// TwinCAT 3 PLC project Main
// ProgramVersion: 3.1.4022.1
// libraries:
//   Tc2_ControllerToolbox, * (Beckhoff Automation GmbH)
//   Tc2_Standard, * (Beckhoff Automation GmbH)
//   Tc2_System, * (Beckhoff Automation GmbH)
//   Tc3_Module, * (Beckhoff Automation GmbH)
//   VisuDialogs, * (System)
// project tree:
//   DUTs/ ST_HISTORY.TcDUT, ST_POINT.TcDUT
//   / GlobalTextList.TcGTLO, PlcTask.TcTTO, Visualization Manager.TcVMO (not stored)
//   GVLs/ Global.TcGVL, Global_Constant.TcGVL
//   GVLs/IO/ IO_Inputs.TcGVL, IO_Outputs.TcGVL
//   POUs/ FB_HeaterCtrl.TcPOU, MAIN.TcPOU, UpdateHistory.TcPOU, InitPidParams.TcPOU
//   VISUs/ VIS_HEATER_CONTROL.TcVIS
// real-time tasks:
//   TASK StandardTask: cycle T#10ms, priority 1, ADS port 350
//   TASK PlcTask: cycle T#10ms, priority 20, ADS port 351
// variable links:
//   Main/Main Instance <-> Simulation/Simulation Instance
//     PlcTask Inputs/IO_Inputs.i_HtrTemp <-> PlcTask Outputs/IO_Outputs.o_HtrTemp
//     PlcTask Outputs/IO_Outputs.o_HtrON <-> PlcTask Inputs/IO_Inputs.i_HtrON
//     PlcTask Outputs/IO_Outputs.o_Restart <-> PlcTask Inputs/IO_Inputs.i_Restart

CONFIGURATION Main
    RESOURCE PLC ON TwinCAT3
        TASK PlcTask(INTERVAL := T#10ms, PRIORITY := 20);
        PROGRAM MAIN WITH PlcTask : MAIN;
    END_RESOURCE
END_CONFIGURATION

// ---- DUTs/ST_HISTORY.TcDUT
// History data
//
TYPE ST_HISTORY:
STRUCT
	
	// Members...
	arPower:       ARRAY[ 1..NUM_HISTORY_POINTS ] OF REAL; // Power history [%]
	arTemperature: ARRAY[ 1..NUM_HISTORY_POINTS ] OF REAL; // Temperature history [°C]
	arTempDiff:    ARRAY[ 1..NUM_HISTORY_POINTS ] OF REAL; // Temp. differences to setp. [°C]
	
END_STRUCT
END_TYPE

// ---- DUTs/ST_POINT.TcDUT
// Point data
//
TYPE ST_POINT:
STRUCT
	
	// Members...
	Power:       REAL; // Heating power [%]
	Temperature: REAL; // Temperature [°C]
	
END_STRUCT
END_TYPE

// ---- GVLs/Global.TcGVL
// Global members
//
VAR_GLOBAL

	// Structures...
	gstHistory: ST_HISTORY; // History data
	
	// Enums...
	gePidState: E_CTRL_STATE; // PID controller state

	// Other global members	
	gPower:    LREAL;      // Heating power [%]
	gSetpoint: REAL := 50; // Temperature setpoint [°C]
	gStepChange: REAL := 10; // Change of auto-step
	gAutoStepTimer: REAL := 0; // Auto-step timer
	gBoolAutoStep: BOOL := FALSE; //Auto-step boolean on/off for auto-step-button
	
END_VAR

// ---- GVLs/Global_Constant.TcGVL
// Global constants
//
VAR_GLOBAL CONSTANT

	// Global constants...
	NUM_HISTORY_POINTS: INT := 120; // Amount of history points
	
END_VAR

// ---- GVLs/IO/IO_Inputs.TcGVL
{attribute 'qualified_only'}
// I/O Inputs
//
VAR_GLOBAL

	// Input signals...
	i_HtrTemp AT %I*: REAL; // Heater temperature [°C]
 
END_VAR

// ---- GVLs/IO/IO_Outputs.TcGVL
{attribute 'qualified_only'}
// I/O Outputs
//
VAR_GLOBAL

	// Output signals...
	o_HtrON   AT %Q*: BOOL; // Heater to ON
	o_Restart AT %Q*: BOOL; // Restart simulation
	o_AddTemp20  AT %Q*: BOOL; // Increase temperature 20C
	o_DropTemp20 AT %Q*: BOOL; // Decrease temperature 20C
	o_AutoStep AT %Q*: BOOL; // Auto-step on/off
 
END_VAR

// ---- POUs/MAIN.TcPOU
// Application main function
//
PROGRAM MAIN
VAR

	// Function blocks...
	fbHeaterCtrl: FB_HeaterCtrl; // Heater control
	
	// Other members...
	Cntr: DINT; // Counter, visiting times
	Step: SINT; // Step counter (1...100)
	
END_VAR

// Update counter
Cntr := ( Cntr + 1 );

// Hasn't the step counter overflowed yet ?
IF Step < 100 THEN

	// Increase the step counter
	Step := ( Step + 1 );
	
// else, Maximum value reached already
ELSE

	// Restart the step counter
	Step := 1;
	
END_IF

// Call the heater control
fbHeaterCtrl( Step := Step );

// Update history
UpdateHistory( Step );

END_PROGRAM

// ---- POUs/FB_HeaterCtrl.TcPOU
// Controls the heater
//
FUNCTION_BLOCK FB_HeaterCtrl
VAR_INPUT
	
	Step: SINT; // Step counter (1...100)
	
END_VAR
VAR
	
	// Function blocks...
	fbPID: FB_CTRL_PID; // PID controller
	
	// Structures...
	stParams: ST_CTRL_PID_PARAMS; // PID controller parameters
	
	// Booleans...
	bInitialized: BOOL; // Initialized
	bRestart:     BOOL; // Restart
	bAutoStep:    BOOL; // Auto-step
	
END_VAR

// Initialize members
bRestart    := ( bRestart    OR IO_Outputs.o_Restart );

// First visit ? 
IF NOT bInitialized THEN
	
	// Initialize PID controller parameters
	bInitialized := TRUE;
	InitPidParams( ADR( stParams ));
	
	bAutoStep := FALSE;
	
END_IF

// Is the the starting step ?
IF Step = 1 THEN
  
	// Update the PID controller once per every second
	fbPID
	(
		fSetpointValue := gSetpoint,
		fActualValue   := IO_Inputs.i_HtrTemp,
		fManSyncValue  := 0,
		bSync          := FALSE,
		eMode          := SEL( bRestart, eCTRL_MODE_ACTIVE, eCTRL_MODE_RESET ),
		bHold          := FALSE,
		stParams       := stParams,
		fOut           => gPower,
		eState         => gePidState
(*
		bARWactive     => BOOL;
		eErrorId       => E_CTRL_ERRORCODES;
		bError         => BOOL;
*)
	);

	// Control the heater to ON/OFF
	IO_Outputs.o_HtrON := ( fbPID.fOut >= Step );
	bRestart           := FALSE;
	
	// Auto-step control
	IF bAutoStep THEN
		gAutoStepTimer := gAutoStepTimer+1;
		IF (gAutoStepTimer >= 20) THEN
			gSetpoint := gSetpoint + gStepChange;
			IF (gSetpoint > 200) THEN
				gSetpoint := 190;
				gStepChange := -10;
			ELSIF (gSetpoint < 0) THEN
				gSetpoint := 10;
				gStepChange := 10;
			END_IF
			gAutoStepTimer := 0;
		END_IF
	END_IF
	
// else, Not the first step now => Is heater controlled to ON ?
ELSIF IO_Outputs.o_HtrON THEN
	
	// Control the heater to ON/OFF
	IO_Outputs.o_HtrON := ( fbPID.fOut >= Step );
	
END_IF

IF IO_Outputs.o_AddTemp20 THEN
	
	gSetpoint := gSetpoint + 20;
	
	IF (gSetpoint > 200) THEN
		gSetpoint := 200;
	END_IF
	
	IO_Outputs.o_AddTemp20 :=FALSE;
	
END_IF

IF IO_Outputs.o_DropTemp20 THEN
	
	gSetpoint := gSetpoint - 20;
	
	IF (gSetpoint < 0) THEN
		gSetpoint := 0;
	END_IF
	
	IO_Outputs.o_DropTemp20 :=FALSE;
	
END_IF

IF IO_Outputs.o_AutoStep THEN
	
	IF bAutoStep THEN
		gStepChange := 10;
		gAutoStepTimer := 0;
		bAutoStep := FALSE;
		gBoolAutoStep := FALSE;
	ELSE
		bAutoStep := TRUE;
		gBoolAutoStep := TRUE;
	END_IF
	
	IO_Outputs.o_AutoStep :=FALSE;
	
END_IF

END_FUNCTION_BLOCK

// ---- POUs/InitPidParams.TcPOU
// Initializes PID controller parameters
//
FUNCTION InitPidParams: BOOL
VAR_INPUT
	
	pstParams: POINTER TO ST_CTRL_PID_PARAMS; // Pointer to PID controller parameters
	
END_VAR

// Initialize the parameters
pstParams^.bARWOnIPartOnly     := FALSE;  // FALSE = the integration of the I-component is halted if the complete controller output reaches the upper or lower limit. TRUE = the integration is halted if the I-component (the output of the integrator) reaches some limit. 
pstParams^.bDInTheFeedbackPath := FALSE;  // Input value OF the internal D-element can be selected with this input 
pstParams^.bPInTheFeedbackPath := FALSE;  // Input value OF the internal P-element can be selected with this input 
pstParams^.fOutMaxLimit        := 100.0;  // Upper limit at which integration is halted and to which the output is limited (ARW measure). Reaching this limit is indicated by a TRUE at the bARWActive output. 
pstParams^.fOutMinLimit        := 0.0;    // Lower limit at which integration is halted and to which the output is limited (ARW measure). Reaching this limit is indicated by a TRUE at the bARWActive output. 
pstParams^.tCtrlCycleTime      := T#1S;   // Cycle time with which the control loop is processed. This must be greater than or equal to TaskCycleTime.
pstParams^.tTaskCycleTime      := T#1S;   // Cycle time with which the function block is called
// PID settings
pstParams^.fKp                 := 2.5;    // Controller amplification / controller coefficient
pstParams^.tTn                 := T#30S;  // Integral action time. The I-component is deactivated if this is parameterized as T#0S. 
pstParams^.tTv                 := T#10S;  // Derivative action time. The D-component is deactivated if this is parameterized as T#0S. 
pstParams^.tTd                 := T#50MS; // Damping time

END_FUNCTION

// ---- POUs/UpdateHistory.TcPOU
// Updates history curve
//
FUNCTION UpdateHistory: BOOL
VAR_INPUT
	
	Step: DINT; // Step counter (1...100)
	
END_VAR
VAR
	
	// Members...
	Index: INT; // Index of history point
	
END_VAR

//
IF Step <> 1 THEN

	RETURN;
	
END_IF

// Scan history data
FOR Index := NUM_HISTORY_POINTS TO 2 BY -1 DO

	//
	gstHistory.arPower[ Index ]       := gstHistory.arPower[ Index - 1 ];
	gstHistory.arTemperature[ Index ] := gstHistory.arTemperature[ Index - 1 ];
	gstHistory.arTempDiff[ Index ]    := gstHistory.arTemperature[ Index ] - gSetpoint;
	
END_FOR 

// Update newest data to history
gstHistory.arPower[ 1 ]       := LREAL_TO_REAL( gPower );
gstHistory.arTemperature[ 1 ] := IO_Inputs.i_HtrTemp;
gstHistory.arTempDiff[ 1 ]    := gstHistory.arTemperature[ 1 ] - gSetpoint;

END_FUNCTION

// ---- GlobalTextList.TcGTLO
TEXTLIST GlobalTextList
  204 = '+20C'
  753 = '-20C'
  104 = 'Admin'
  481 = 'Auto-step'
  413 = 'Controller amplification Kp: %.1f'
  343 = 'Controller amplification [Kp]: %.1f'
  741 = 'Controller amplification [Kp]: %.1f '
  821 = 'Derivative action time Tv: %s'
  682 = 'Derivative action time [Tv]: %s'
  494 = 'Derivative action time [Tv]: %s '
  373 = 'gAutoStepTimer'
  534 = 'Global.gAutoStepTimer'
  637 = 'Heating Power %.1f %'
  88 = 'Increase 20C'
  263 = 'Integral action time Tn: %s'
  214 = 'Integral action time [Tn]: %s'
  982 = 'Integral action time [Tn]: %s '
  572 = 'Kp %.1f'
  352 = 'None'
  603 = 'Operator'
  417 = 'PID controller state: %s'
  785 = 'Power %.1f %'
  26 = 'Power [%]'
  804 = 'Restart'
  212 = 'Service'
  34 = 'Setpoint %.1f °C'
  679 = 'Td %.1f'
  938 = 'Td %s'
  202 = 'Temperature %.1f °C'
  262 = 'Temperature [°C]'
  159 = 'Tn %s'
  557 = 'Tv %s'
END_TEXTLIST

// ---- VISUs/VIS_HEATER_CONTROL.TcVIS
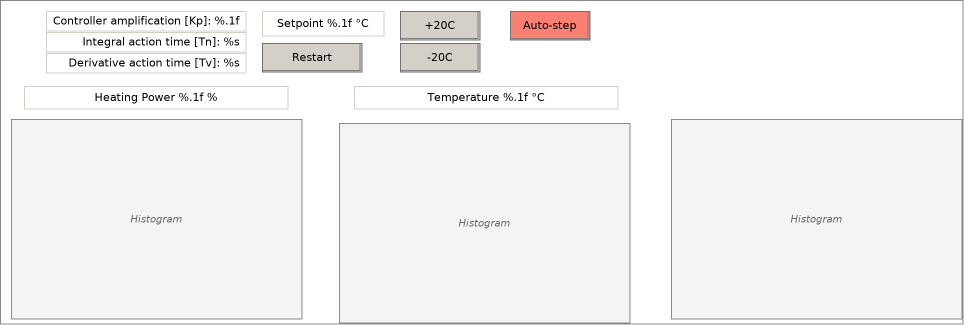
VISUALIZATION VIS_HEATER_CONTROL  // 964x325
    Histogram (11,119 291x200), scale format: %.1f, scale 0..100
        p1518820177: gstHistory.arPower
        p102497268: gstHistory.arPower
        p788070771: ARRAY [1..NUM_HISTORY_POINTS] OF REAL
    Histogram (339,123 291x200), scale format: %.1f, scale 0..200
        p1518820177: gstHistory.arTemperature
        p102497268: gstHistory.arTemperature
        p788070771: ARRAY [1..NUM_HISTORY_POINTS] OF REAL
    Textfield (24,86 264x23), "Heating Power %.1f %", text variable: gPower
    Textfield (354,86 264x23), "Temperature %.1f °C", text variable: IO_Inputs.i_HtrTemp
    Textfield (262,11 122x25), "Setpoint %.1f °C", text variable: gSetpoint
        OnMouseClick: write the text variable via Default
    Textfield (46,53 200x20), "Derivative action time [Tv]: %s", text variable: MAIN.fbHeaterCtrl.stParams.tTv
        OnMouseClick: write the text variable via Default
    Button (262,43 100x29), "Restart"
        tap IO_Outputs.o_Restart
    Textfield (46,32 200x20), "Integral action time [Tn]: %s", text variable: MAIN.fbHeaterCtrl.stParams.tTn
        OnMouseClick: write the text variable via Default
    Textfield (46,11 200x20), "Controller amplification [Kp]: %.1f", text variable: MAIN.fbHeaterCtrl.stParams.fKp
        OnMouseClick: write the text variable via Default
    Button (400,11 80x29), "+20C"
        tap IO_Outputs.o_AddTemp20
    Button (400,43 80x29), "-20C"
        tap IO_Outputs.o_DropTemp20
    Histogram (671,119 291x200), scale format: %.1f, scale -5..5
        p1518820177: gstHistory.arTempDiff
        p102497268: gstHistory.arTempDiff
        p788070771: ARRAY [1..NUM_HISTORY_POINTS] OF REAL
    Button (510,11 80x29), "Auto-step", colour toggle: gBoolAutoStep
        tap IO_Outputs.o_AutoStep
END_VISUALIZATION
